{attribute 'qualified_only'}
{attribute 'strict'}
{attribute 'to_string'}
TYPE PROBLEM_HANDLING_RESULT :
(
	SET_ERROR_AND_STOP_COMPONENT,
	SET_ERROR,
	IGNORE
);
END_TYPE

(* stored: Version 1.1.0.1
   DUT PROBLEM_HANDLING_RESULT: Id {1aa00b00-e88d-42e5-af75-9579a4cfa4a2} *)
